// TIA Portal V17 export
// export: Created 2022-07-28T18:02:45.0837111Z, ExportSetting None, DisplayName Totally Integrated Automation Portal, DisplayVersion V17, DisplayName TIA Portal Openness, DisplayVersion V17, DisplayName TIA Portal Teamcenter Gateway, DisplayVersion V17, DisplayName TIA Portal Version Control Interface, DisplayVersion V17, DisplayName TIA Portal Test Suite Advanced, DisplayVersion V17, DisplayName SINAMICS Startdrive Advanced, DisplayVersion V17, DisplayName SINAMICS DCC, DisplayVersion V17, DisplayName SINAMICS Startdrive G130, G150, S120, S150, SINAMICS MV, S210, DisplayVersion V17, DisplayName SINAMICS Startdrive G110M, G120, G120C, G120D, G120P, G115D, DisplayVersion V17, DisplayName STEP 7 Professional, DisplayVersion V17, DisplayName SIMATIC Energy Suite, DisplayVersion V17, DisplayName STEP 7 CFC, DisplayVersion V17, DisplayName STEP 7 Safety, DisplayVersion V17, DisplayName WinCC Advanced / Unified PC, DisplayVersion V17, DisplayName SIMATIC Visualization Architect, DisplayVersion V17
FUNCTION "Lib_FC_Auto" : Void   // FC8, SCL
{ S7_Optimized_Access := 'TRUE' }
// stored: SetENOAutomatically false
   VAR_INPUT
      IB_Initialisation : Bool;   // 1 = "FirstScan" / Стартова ініціалізація/Restart PLC is active
   END_VAR
   VAR_IN_OUT
      IOs_AutoControl : "Lib_UDT_AutoControl";
   END_VAR
   VAR_TEMP
      ts_AutoControl : "Lib_UDT_AutoControl";
   END_VAR
BEGIN
   // REGION Стартова Ініціалізація AutoControl
   //--------------------------------------
   //Reset #ts_AutoControl <- "DB_AutoControl_arr".AutoControl_arr[999];
   #ts_AutoControl := #IOs_AutoControl;
   //--------------------------------------
   //-------------------------------------
   IF #IB_Initialisation THEN
       #ts_AutoControl.CTW.%B0 := 2#00000000;
       #ts_AutoControl.CTW.%B1 := 2#00000000;
       #ts_AutoControl.CTW.%B2 := #ts_AutoControl.CTW.%B2 AND 2#10000000;
       #ts_AutoControl.CTW.%B3 := 2#00000000;
       #ts_AutoControl.Global_CMD := 1;//MANREM - Перевести в ManualRemote -ручний HMI
   END_IF;
   //-------------------------------------
   //AutoControl
   //CTW.%X0:= CmdAutoOpen - (Static bit)
   //CTW.%X1:= CmdAutoClose - (Static bit)
   //////CTW.%X2:=
   //////CTW.%X3:=
   //////CTW.%X4:=
   //////CTW.%X6:=
   //////CTW.%X7:=
   //////CTW.%X8:=
   //////CTW.%X9:=
   //////CTW.%X10:=
   //////CTW.%X11:=
   //////CTW.%X12:=
   //////CTW.%X13:=
   //////CTW.%X14:=
   //////CTW.%X15:=
   //////CTW.%X16:= go to ManualRemote - (resetable bit)
   //////CTW.%X17:= go to Auto - (resetable bit)
   //////CTW.%X18:= go to ManualLocal - (resetable bit)
   //////CTW.%X19:= ON Simulation - (resetable bit)
   //////CTW.%X20:= OFF Simulation - (resetable bit)
   //////CTW.%X21:= 
   //////CTW.%X22:= go to Disable - (resetable bit)
   //////CTW.%X23:= Independent - (Static bit)
   //////CTW.%X24:=
   //////CTW.%X25:=
   //////CTW.%X26:=
   //////CTW.%X27:=
   //////CTW.%X28:=
   //////CTW.%X29:=
   //////CTW.%X30:=
   //////CTW.%X31:=
   //-------------------------------------
   //Get data from general DB of Auto, Inverter for exchange data between diff modules one object

   REGION CMD 
       IF #ts_AutoControl.Global_CMD > 0
           AND #ts_AutoControl.Global_CMD < 200 THEN
           CASE #ts_AutoControl.Global_CMD OF
               3, 4, 5, 6:// заблоковані командт
                   #ts_AutoControl.Global_CMD := 0;
               100..131: // Reset bit CTW
                   #ts_AutoControl.CTW := ROR(IN := #ts_AutoControl.CTW, N := #ts_AutoControl.Global_CMD - 100);
                   #ts_AutoControl.CTW.%X0 := FALSE;
                   #ts_AutoControl.CTW := ROL(IN := #ts_AutoControl.CTW, N := #ts_AutoControl.Global_CMD - 100);
                   #ts_AutoControl.Global_CMD := 0;

               150..181: // Set bit CTW
                   #ts_AutoControl.CTW := ROR(IN := #ts_AutoControl.CTW, N := #ts_AutoControl.Global_CMD - 150);
                   #ts_AutoControl.CTW.%X0 := TRUE;
                   #ts_AutoControl.CTW := ROL(IN := #ts_AutoControl.CTW, N := #ts_AutoControl.Global_CMD - 150);
                   #ts_AutoControl.Global_CMD := 0;
                   // 164..195: // invert bit CTW
                   //     #ts_AutoControl.CTW := ROR(IN := #ts_AutoControl.CTW, N := #ts_AutoControl.Global_CMD - 164);
                   //     #ts_AutoControl.CTW.%X0 := NOT #ts_AutoControl.CTW.%X0;
                   //     #ts_AutoControl.CTW := ROL(IN := #ts_AutoControl.CTW, N := #ts_AutoControl.Global_CMD - 164);
                   //     #ts_AutoControl.Global_CMD := 0;
               ELSE
                   ;
           END_CASE;


       END_IF;


   END_REGION
   // ---------------------------------------------------------------

   REGION - CTW - >  to -> Global CMD ///////From auto array CTW_BIT
       (*Motor MODE - CMD From auto array db*)
       // IF #ts_AutoControl.Global_CMD = 0 AND
       //     BYTE_TO_INT(#ts_AutoControl.CTW.%B2 AND 2#01111111) <> 0 THEN
       //     CASE BYTE_TO_INT(#ts_AutoControl.CTW.%B2 AND 2#01111111) OF
       //         1:  (*bit 0 Manual =  Function change to Manual mode - активує ManualRemote*)
       //             #ts_AutoControl.Global_CMD := 1;
       //         2:  (*bit 1 AUTO = Auto Function change to Auto mode*)
       //             #ts_AutoControl.Global_CMD := 2;
       //             //4:  (*bit 2 Перевести в ManualLocal - ручний зі щита кнопками*)
       //             //    #ts_AutoControl.Global_CMD := 3;
       //         8:  (*bit 3 Simulation - ON Симуляція*)
       //             #ts_AutoControl.Global_CMD := 7;
       //         16:  (*bit 4 Simulation - OFF Симуляція*)
       //             #ts_AutoControl.Global_CMD := 8;
       //             //32: (*bit 5 DSABLE/OFF/STOP*)
       //             //    ;
       //         64:  (*bit 6 DSABLE/OFF/STOP*)
       //             #ts_AutoControl.Global_CMD := 10;
       //         ELSE  // Statement section ELSE
       //             #ts_AutoControl.Global_CMD := 0;
       //     END_CASE;
       //     #ts_AutoControl.CTW.%B2 :=#ts_AutoControl.CTW.%B2 AND 2#10000000;
       // END_IF;
   END_REGION




   #ts_AutoControl.CTW.%X23 := TRUE;

   //---------------------------------------------------------------
   #IOs_AutoControl := #ts_AutoControl;
END_FUNCTION
